{attribute 'TcGenerated'}
// This function has been automatically generated from the project information.
VAR_GLOBAL CONSTANT
	{attribute 'const_non_replaced'}
	{attribute 'linkalways'}
	stLibVersion_MBC_TC3_PCS_Library : ST_LibVersion := (iMajor := 1, iMinor := 0, iBuild := 0, iRevision := 2, sVersion := '1.0.0.2');
END_VAR

(* stored: Version 1.1.0.1, ProductVersion 3.1.4022.10
   GVL Global_Version: Id {b04f62c3-23a7-0bc4-3d46-52acd3064e70} *)
